FUNCTION_BLOCK Plant (* Basic Function Block Type *)
  (* Standard: 61499-2 *)
  (* Version 0.0, 4/23/2019, vshatrov, nxtControl GmbH, Template *)
  PACKAGE Main;
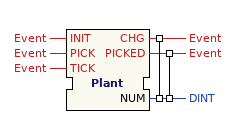
  EVENT_INPUT
    INIT; (* Initialization Request *)
    PICK; (* Normal Execution Request *)
    TICK;
  END_EVENT
  EVENT_OUTPUT
    CHG WITH NUM; (* Execution Confirmation *)
    PICKED WITH NUM;
  END_EVENT
  VAR_OUTPUT
    NUM : DINT; (* Output event qualifier *)
  END_VAR
  VAR
    current : DINT;
  END_VAR
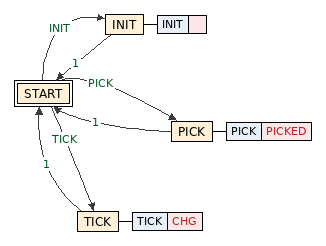
  EC_STATES
    START; (* Initial State *)
    INIT : INIT; (* Initialization *)
    TICK : TICK -> CHG; (* Normal execution *)
    PICK : PICK -> PICKED;
  END_STATES
  EC_TRANSITIONS
    START TO INIT := INIT;
    INIT TO START := 1;
    START TO TICK := TICK;
    TICK TO START := 1;
    START TO PICK := PICK;
    PICK TO START := 1;
  END_TRANSITIONS
  ALGORITHM INIT IN ST: (* Initialization algorithm *)
current := 0;
  END_ALGORITHM
  ALGORITHM TICK IN ST: (* Normally executed algorithm *)
current := (current + 1) MOD 10;
NUM := current;
  END_ALGORITHM
  ALGORITHM PICK IN ST:
NUM := current;
  END_ALGORITHM
END_FUNCTION_BLOCK
